// TIA Portal V19 export
FUNCTION "CarriageLub_CALL" : Void   // FC168, LAD
TITLE = Carriage Lubrication CALL
// stored: SetENOAutomatically false
BEGIN

REGION Network 1: Carriage Slide lubrication >>>
END_REGION

REGION Network 2: Dispenser valve Data In
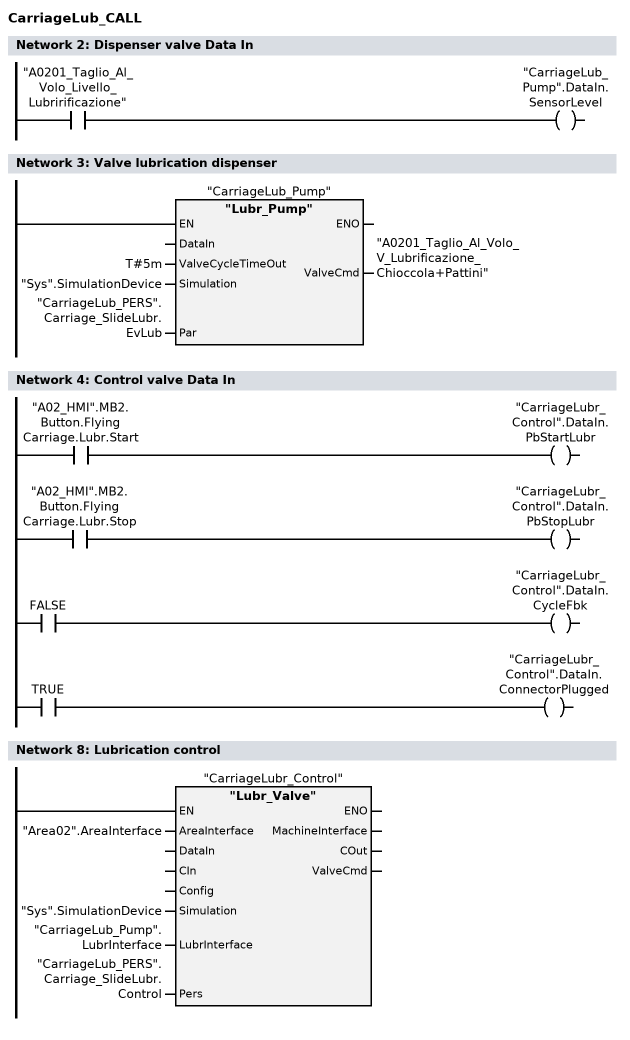
   RUNG wire#powerrail
      Contact( "A0201_Taglio_Al_Volo_Livello_Lubririficazione" )
      Coil( "CarriageLub_Pump".DataIn.SensorLevel )
   END_RUNG
   // the same network as SCL:
   "CarriageLub_Pump".DataIn.SensorLevel := "A0201_Taglio_Al_Volo_Livello_Lubririficazione";
END_REGION

REGION Network 3: Valve lubrication dispenser
   RUNG wire#powerrail
      "CarriageLub_Pump"(DataIn :=, ValveCycleTimeOut := T#5m, Simulation := "Sys".SimulationDevice, Par := "CarriageLub_PERS".Carriage_SlideLubr.EvLub, ValveCmd => "A0201_Taglio_Al_Volo_V_Lubrificazione_Chioccola+Pattini")
   END_RUNG
   // the same network as SCL:
   "CarriageLub_Pump"(ValveCycleTimeOut := T#5m,   // "Lubr_Pump"
                      Simulation := "Sys".SimulationDevice,
                      Par := "CarriageLub_PERS".Carriage_SlideLubr.EvLub,
                      ValveCmd => "A0201_Taglio_Al_Volo_V_Lubrificazione_Chioccola+Pattini");
END_REGION

REGION Network 4: Control valve Data In
   RUNG wire#powerrail
      Contact( "A02_HMI".MB2.Button.FlyingCarriage.Lubr.Start )
      Coil( "CarriageLubr_Control".DataIn.PbStartLubr )
   END_RUNG
   RUNG wire#powerrail
      Contact( "A02_HMI".MB2.Button.FlyingCarriage.Lubr.Stop )
      Coil( "CarriageLubr_Control".DataIn.PbStopLubr )
   END_RUNG
   RUNG wire#powerrail
      Contact( FALSE )
      Coil( "CarriageLubr_Control".DataIn.CycleFbk )
   END_RUNG
   RUNG wire#powerrail
      Contact( TRUE )
      Coil( "CarriageLubr_Control".DataIn.ConnectorPlugged )
   END_RUNG
   // the same network as SCL:
   "CarriageLubr_Control".DataIn.PbStartLubr := "A02_HMI".MB2.Button.FlyingCarriage.Lubr.Start;
   "CarriageLubr_Control".DataIn.PbStopLubr := "A02_HMI".MB2.Button.FlyingCarriage.Lubr.Stop;
   "CarriageLubr_Control".DataIn.CycleFbk := FALSE;
   "CarriageLubr_Control".DataIn.ConnectorPlugged := TRUE;
END_REGION

REGION Network 5 (SCL): Valve Cin
   "CarriageLubr_Control".CIn.LubrEnable := NOT "FlyingCarriage".COut.Standstill;
   "CarriageLubr_Control".CIn.ActualPosition := "FlyingCarriage".Ax.AxisSts.ActualPosition;
   "CarriageLubr_Control".CIn.OperationDone := FALSE;
END_REGION

REGION Network 6 (SCL): Valve Config
   "CarriageLubr_Control".Config.WorkMode :=2;
   "CarriageLubr_Control".Config.CounterMode := 0;
   "CarriageLubr_Control".Config.ValveType := 0;
   "CarriageLubr_Control".Config.ManualCmdTimeOut := T#20M;
END_REGION

REGION Network 7 (SCL): Distance meter reset
   IF "CarriageLub_PERS".CarriageLub_Pers_HMI_ResetCounter
   THEN
       "CarriageLub_PERS".Carriage_SlideLubr.Control.LubrReqCounter := 0.0;
       "CarriageLub_PERS".CarriageLub_Pers_HMI_ResetCounter := FALSE;
   END_IF;
END_REGION

REGION Network 8: Lubrication control
   RUNG wire#powerrail
      "CarriageLubr_Control"(AreaInterface := "Area02".AreaInterface, DataIn :=, CIn :=, Config :=, Simulation := "Sys".SimulationDevice, LubrInterface := "CarriageLub_Pump".LubrInterface, Pers := "CarriageLub_PERS".Carriage_SlideLubr.Control, MachineInterface =>, COut =>, ValveCmd =>)
   END_RUNG
   // the same network as SCL:
   "CarriageLubr_Control"(AreaInterface := "Area02".AreaInterface,   // "Lubr_Valve"
                          Simulation := "Sys".SimulationDevice,
                          LubrInterface := "CarriageLub_Pump".LubrInterface,
                          Pers := "CarriageLub_PERS".Carriage_SlideLubr.Control);
END_REGION
END_FUNCTION
